PROGRAM MAIN
VAR
	i: INT;
END_VAR

i := i + 1;

END_PROGRAM

(* stored: Version 1.1.0.1, ProductVersion 3.1.4024.11
   POU MAIN: Id {6b5c19e2-6669-4ea9-ab48-1e2aa828cb18}, SpecialFunc None *)
